TEXTLIST AkCmbTxtList
  1 = '1'
  2 = '2'
  3 = '3'
  4 = '4'
   = ''
END_TEXTLIST

(* stored: Version 1.1.0.1, ProductVersion 3.1.4024.4
   TextList AkCmbTxtList: Id {ef0c3b59-0479-4b5c-b299-ed8fe5ba8ded} *)
